INTERFACE I_Line_Builder EXTENDS T_Query_Interface

END_INTERFACE

(* stored: Version 1.1.0.1, ProductVersion 3.1.4024.4
   Itf I_Line_Builder: Id {25de0b71-969b-4988-a3f7-e3b24d80f633} *)
